# EPICS substitutions: src/iocdoc/testfiles/iocBoot/ioc495idc/templates/motor.substitutions
file "$(MOTOR)/databases/motor.db"
{
pattern
{P,      M,     DTYP,        C,  S,  DESC,          EGU, DIR,  VELO,  VBAS,  ACCL,  BDST,  BVEL,  BACC,  MRES,  PREC,  DHLM,  DLLM,  INIT}
# NES
{495idc:, "m1",  "OMS MAXv",  0,  0,  "motor 1",  mm,  Pos,  1,     .1,    .2,	 0,   1,     .2,    0.01,  5,	  100,   -100,  "LH"}
{495idc:, "m2",  "OMS MAXv",  0,  1,  "motor 2",  mm,  Pos,  1,     .1,    .2,	 0,   1,     .2,    0.01,  5,	  100,   -100,  "LH"}
{495idc:, "m3",  "OMS MAXv",  0,  2,  "motor 3",  mm,  Pos,  1,     .1,    .2,	 0,   1,     .2,    0.01,  5,	  100,   -100,  "LH"}
{495idc:, "m4",  "OMS MAXv",  0,  3,  "motor 4",  mm,  Pos,  1,     .1,    .2,	 0,   1,     .2,    0.01,  5,	  100,   -100,  "LH"}
{495idc:, "m5",  "OMS MAXv",  0,  4,  "motor 5",  mm,  Pos,  1,     .1,    .2,	 0,   1,     .2,    0.01,  5,	  100,   -100,  "LH"}
{495idc:, "m6",  "OMS MAXv",  0,  5,  "motor 6",  mm,  Pos,  1,     .1,    .2,	 0,   1,     .2,    0.01,  5,	  100,   -100,  "LH"}
{495idc:, "m7",  "OMS MAXv",  0,  6,  "motor 7",  mm,  Pos,  1,     .1,    .2,	 0,   1,     .2,    0.01,  5,	  100,   -100,  "LH"}
{495idc:, "m8",  "OMS MAXv",  0,  7,  "motor 8",  mm,  Pos,  1,     .1,    .2,	 0,   1,     .2,    0.01,  5,	  100,   -100,  "LH"}
# DET
{495idc:, "m9",  "OMS MAXv",  1,  0,  "motor  9",  mm,  Pos,  1,     .1,    .2,    0,   1,     .2,    0.01,  5,     100,   -100,  "LH"}
{495idc:, "m10", "OMS MAXv",  1,  1,  "motor 10",  mm,  Pos,  1,     .1,    .2,    0,   1,      .2,    0.01,  5,     100,   -100,  "LH"}
{495idc:, "m11", "OMS MAXv",  1,  2,  "motor 11",  mm,  Pos,  1,     .1,    .2,    0,   1,      .2,    0.01,  5,     100,   -100,  "LH"}
{495idc:, "m12", "OMS MAXv",  1,  3,  "motor 12",  mm,  Pos,  1,     .1,    .2,    0,   1,      .2,    0.01,  5,     100,   -100,  "LH"}
{495idc:, "m13", "OMS MAXv",  1,  4,  "motor 13",  mm,  Pos,  1,     .1,    .2,    0,   1,      .2,    0.01,  5,     100,   -100,  "LH"}
{495idc:, "m14", "OMS MAXv",  1,  5,  "motor 14",  mm,  Pos,  1,     .1,    .2,    0,   1,      .2,    0.01,  5,     100,   -100,  "LH"}
{495idc:, "m15", "OMS MAXv",  1,  6,  "motor 15",  mm,  Pos,  1,     .1,    .2,    0,   1,      .2,    0.01,  5,     100,   -100,  "LH"}
{495idc:, "m16", "OMS MAXv",  1,  7,  "motor 16",  mm,  Pos,  1,     .1,    .2,    0,   1,      .2,    0.01,  5,     100,   -100,  "LH"}
}
#	# DET m9-10
#	file "$(TOP)/495idcApp/Db/soft_pzt_motor.db"
#	{
#	pattern
#	{P,      N,  M, DAC}
#	{495idc:, 17, m, DAC1_1}
#	{495idc:, 18, m, DAC1_2}
#	}
# DET m11-12
file "$(MOTOR)/databases/asyn_motor.db"
{
pattern
{P,      N,  M,     DTYP,	 PORT,  ADDR,  DESC,		EGU,	DIR,   VELO,	VBAS,	ACCL,	BDST,	BVEL,	BACC,	MRES,	SREV,	UREV,	PREC,	DHLM,	DLLM,	INIT}
{495idc:, 19, "m19", asynMotor,   IA1,	0,     "motor 19",	mm,	Pos,   1,	0.1,	.2,	0,	1,	.2,	0.001,  1,	.001,	3,	400,	0,	""}
{495idc:, 20, "m20", asynMotor,   IA1,	2,     "motor 20",	mm,	Pos,   1,	0.1,	.2,	0,	1,	.2,	0.001,  1,	.001,	3,	400,	0,	""}
}
#	# DET m13-14
#	file "$(TOP)/495idcApp/Db/asyn_slave_motor.db"
#	{
#	pattern
#	{P,      M,	 F,	DTYP,		PORT,  AXIS,	CMD,	    DESC,		PREC,	EGU,	MSTR}
#	{495idc:, m21:,   pos	asynFloat64,	IA1,   1,	POSITION    "slave motor pos",  4	mm	m19}
#	{495idc:, m22:,   pos	asynFloat64,	IA1,   3,	POSITION    "slave motor pos",  4	mm	m20}
#	}
